// TwinCAT 3 PLC project sACN_PLC
// ProgramVersion: 3.1.4026.18
// libraries:
//   Tc2_Standard, * (Beckhoff Automation GmbH)
//   Tc2_System, * (Beckhoff Automation GmbH)
//   Tc2_TcpIp, * (Beckhoff Automation GmbH)
//   Tc2_Utilities, * (Beckhoff Automation GmbH)
//   Tc3_EventLogger, * (Beckhoff Automation GmbH)
//   Tc3_sACN, * (Beckhoff Automation GmbH)
// project tree:
//   IO/ IO.TcPOU, Term06.TcPOU, Term07.TcPOU
//   / PlcTask.TcTTO
//   POUs/Case_01/ c01_SimpleUsecase.TcPOU
//   POUs/Case_02/ c02_SharingCommunicator.TcPOU
//   POUs/Case_02/SubProgramms/ PRG_SimpleSending.TcPOU, PRG_SimpleReceiving.TcPOU
//   POUs/Case_03/ c03_InteractingWithIO.TcPOU
//   POUs/Case_04/ c4_MultiuniverseSource.TcPOU
//   POUs/Case_05/ c05_CustomFBs.TcPOU
//   POUs/Case_05/SBSPM Extended POUs/ FB_sACN_ReceiverAndMerger_SBSPM.TcPOU, FB_sACN_Source_SBSPM.TcPOU, ST_ReceivedSourceSBSPM.TcDUT
//   POUs/Case_06/ c06_TrackingEvents.TcPOU, FB_sAcnMessagesCatcher.TcPOU
//   POUs/ MAIN.TcPOU
// real-time tasks:
//   TASK PlcTask: cycle T#10ms, priority 20, ADS port 350
// I/O:
//   DEVICE Device 1 (EtherCAT) (disabled), AmsNetId 172.17.152.255.2.1
//     Term 1 (EK1200) [EK1200-5000 EtherCAT Power supply (2A E-Bus)]
//       Term 2 (EK1110) [EK1110 EtherCAT extension]
//     Term 3 (EK1100) [EK1100 EtherCAT Coupler (2A E-Bus)]
//       Term 4 (EL4002) [EL4002 2Ch. Ana. Output 0-10V, 12bit]
//       Term 5 (EL4022) [EL4022 2Ch. Ana. Output 4-20mA, 12bit]
//       Term 6 (EL6851) [EL6851 DMX Master]
//       Term 7 (EL6851-0010) [EL6851-0010 DMX Slave]
//       Term 9 (EL9011) [EL9011 End Terminal]
// variable links:
//   sACN_PLC/sACN_PLC Instance <-> Device 1 (EtherCAT)/Term 3 (EK1100)/Term 6 (EL6851)
//     PlcTask Outputs/Term06.ChannelsLength <-> DMX Control/Channel length
//     PlcTask Outputs/Term06.DmxChannels <-> DMX Channel 1-64/Channel 1
//     PlcTask Outputs/Term06.DmxChannels @bit 72 <-> DMX Channel 1-64/Channel 10
//     PlcTask Outputs/Term06.DmxChannels @bit 80 <-> DMX Channel 1-64/Channel 11
//     PlcTask Outputs/Term06.DmxChannels @bit 88 <-> DMX Channel 1-64/Channel 12
//     PlcTask Outputs/Term06.DmxChannels @bit 96 <-> DMX Channel 1-64/Channel 13
//     PlcTask Outputs/Term06.DmxChannels @bit 104 <-> DMX Channel 1-64/Channel 14
//     PlcTask Outputs/Term06.DmxChannels @bit 112 <-> DMX Channel 1-64/Channel 15
//     PlcTask Outputs/Term06.DmxChannels @bit 120 <-> DMX Channel 1-64/Channel 16
//     PlcTask Outputs/Term06.DmxChannels @bit 8 <-> DMX Channel 1-64/Channel 2
//     PlcTask Outputs/Term06.DmxChannels @bit 16 <-> DMX Channel 1-64/Channel 3
//     PlcTask Outputs/Term06.DmxChannels @bit 24 <-> DMX Channel 1-64/Channel 4
//     PlcTask Outputs/Term06.DmxChannels @bit 32 <-> DMX Channel 1-64/Channel 5
//     PlcTask Outputs/Term06.DmxChannels @bit 40 <-> DMX Channel 1-64/Channel 6
//     PlcTask Outputs/Term06.DmxChannels @bit 48 <-> DMX Channel 1-64/Channel 7
//     PlcTask Outputs/Term06.DmxChannels @bit 56 <-> DMX Channel 1-64/Channel 8
//     PlcTask Outputs/Term06.DmxChannels @bit 64 <-> DMX Channel 1-64/Channel 9
//   sACN_PLC/sACN_PLC Instance <-> Device 1 (EtherCAT)/Term 3 (EK1100)/Term 7 (EL6851-0010)
//     PlcTask Inputs/Term07.DMX_Control_SDX16 <-> DMX Channel 1-64/Channel 1
//     PlcTask Inputs/Term07.DMX_Control_SDX16 @bit 72 <-> DMX Channel 1-64/Channel 10
//     PlcTask Inputs/Term07.DMX_Control_SDX16 @bit 80 <-> DMX Channel 1-64/Channel 11
//     PlcTask Inputs/Term07.DMX_Control_SDX16 @bit 88 <-> DMX Channel 1-64/Channel 12
//     PlcTask Inputs/Term07.DMX_Control_SDX16 @bit 96 <-> DMX Channel 1-64/Channel 13
//     PlcTask Inputs/Term07.DMX_Control_SDX16 @bit 104 <-> DMX Channel 1-64/Channel 14
//     PlcTask Inputs/Term07.DMX_Control_SDX16 @bit 112 <-> DMX Channel 1-64/Channel 15
//     PlcTask Inputs/Term07.DMX_Control_SDX16 @bit 120 <-> DMX Channel 1-64/Channel 16
//     PlcTask Inputs/Term07.DMX_Control_SDX16 @bit 8 <-> DMX Channel 1-64/Channel 2
//     PlcTask Inputs/Term07.DMX_Control_SDX16 @bit 16 <-> DMX Channel 1-64/Channel 3
//     PlcTask Inputs/Term07.DMX_Control_SDX16 @bit 24 <-> DMX Channel 1-64/Channel 4
//     PlcTask Inputs/Term07.DMX_Control_SDX16 @bit 32 <-> DMX Channel 1-64/Channel 5
//     PlcTask Inputs/Term07.DMX_Control_SDX16 @bit 40 <-> DMX Channel 1-64/Channel 6
//     PlcTask Inputs/Term07.DMX_Control_SDX16 @bit 48 <-> DMX Channel 1-64/Channel 7
//     PlcTask Inputs/Term07.DMX_Control_SDX16 @bit 56 <-> DMX Channel 1-64/Channel 8
//     PlcTask Inputs/Term07.DMX_Control_SDX16 @bit 64 <-> DMX Channel 1-64/Channel 9

CONFIGURATION sACN_PLC
    RESOURCE PLC ON TwinCAT3
        TASK PlcTask(INTERVAL := T#10ms, PRIORITY := 20);
        PROGRAM MAIN WITH PlcTask : MAIN;
    END_RESOURCE
END_CONFIGURATION

// ---- POUs/Case_05/SBSPM Extended POUs/ST_ReceivedSourceSBSPM.TcDUT
TYPE ST_ReceivedSourceSBSPM :
STRUCT
	Name 		: STRING(63);
	CID			: Guid;
	Priority	: USINT(0..200);
	IpAddress	: T_IPv4Addr;
	LastFrameNum: USINT;
	SeqErr      : USINT;
	Jumps		: USINT;
	LastPriorities		: ARRAY [1..512] OF USINT;
	LastDMXproperties 	: ARRAY [1..512] OF USINT;
	timeout 	: TON;
END_STRUCT
END_TYPE

// ---- POUs/MAIN.TcPOU
PROGRAM MAIN
VAR
	ChangeValuesTimer : TON;
	i : UINT;
	
	ActiveSample : USINT := 01;
END_VAR

IO();

CASE ActiveSample OF
	01: //<========= CASE 01: Simple Send and Receive sACN Data =========>
		c01_SimpleUsecase();
		
		ChangeValuesTimer(IN:= NOT ChangeValuesTimer.Q, PT:= T#50MS);
		IF ChangeValuesTimer.Q THEN
			FOR i:=1 TO 16 DO
				c01_SimpleUsecase.InDmxData_U111[i] := c01_SimpleUsecase.InDmxData_U111[i] + 1;
				c01_SimpleUsecase.InDmxData_U333[i] := c01_SimpleUsecase.InDmxData_U333[i] - 1;
			END_FOR
		END_IF
	
	02: //<========= CASE 02: Single Communicator, Multiple Subprograms =========>
		c02_SharingCommunicator();
		
	03: //<========= CASE 03: Integration the sACN protocol with hardware DMX terminals =========>
		c03_InteractingWithIO();
		
	04: //<========= CASE 04: Idea for multiuniverse sACN source =========>
		ChangeValuesTimer(IN:= NOT ChangeValuesTimer.Q, PT:= T#50MS);
		
		c4_MultiuniverseSource(	 Enable:= , 
							 SourceName:= 'Sample Multiuniverse Source' ,
									CID:= Tc2_Utilities.STRING_TO_GUID('6f872ff2-8f47-4ea3-a351-549a76e10665')); //Generated by https://www.guidgenerator.com/
									
		IF ChangeValuesTimer.Q THEN
			FOR i:=1 TO 64 DO
				c4_MultiuniverseSource.InDmxData_U111[i] := c4_MultiuniverseSource.InDmxData_U111[i] + 1;
			END_FOR
			FOR i:=1 TO 128 DO
				c4_MultiuniverseSource.InDmxData_U222[i] := c4_MultiuniverseSource.InDmxData_U222[i] - 1;
			END_FOR
			FOR i:=1 TO 256 DO
				c4_MultiuniverseSource.InDmxData_U333[i] := c4_MultiuniverseSource.InDmxData_U333[i] + 1;
			END_FOR
			FOR i:=1 TO 512 DO
				c4_MultiuniverseSource.InDmxData_U444[i] := c4_MultiuniverseSource.InDmxData_U444[i] - 1;
			END_FOR
		END_IF
		
	05: //<========= CASE 05: Castom FB's =========>
		c05_CustomFBs();
END_CASE

//<========= CASE 06: Catching error events =========>
c06_TrackingEvents();

END_PROGRAM

// ---- IO/IO.TcPOU
PROGRAM IO
VAR
END_VAR

Term06();

Term07();

END_PROGRAM

// ---- IO/Term06.TcPOU
//EL6851 Terminal (DMX Master) programm
PROGRAM Term06 
VAR_INPUT
	DmxLightFixture_Left  : ARRAY [1..8] OF USINT;
	DmxLightFixture_Right : ARRAY [1..8] OF USINT;
END_VAR
VAR_OUTPUT
	ChannelsLength	AT %Q*: UINT := 16;
	DmxChannels		AT %Q*: ARRAY [1..16] OF USINT; 
END_VAR

DmxChannels  [1] := DmxLightFixture_Left [1];
DmxChannels  [2] := DmxLightFixture_Left [2];
DmxChannels  [3] := DmxLightFixture_Left [3];
DmxChannels  [4] := DmxLightFixture_Left [4];
                    
DmxChannels  [5] := DmxLightFixture_Left [5];
DmxChannels  [6] := DmxLightFixture_Left [6];
DmxChannels  [7] := DmxLightFixture_Left [7];
DmxChannels  [8] := DmxLightFixture_Left [8];

DmxChannels  [9] := DmxLightFixture_Right [1];
DmxChannels [10] := DmxLightFixture_Right [2];
DmxChannels [11] := DmxLightFixture_Right [3];
DmxChannels [12] := DmxLightFixture_Right [4];
                                                          
DmxChannels [13] := DmxLightFixture_Right [5];
DmxChannels [14] := DmxLightFixture_Right [6];
DmxChannels [15] := DmxLightFixture_Right [7];
DmxChannels [16] := DmxLightFixture_Right [8];

END_PROGRAM

// ---- IO/Term07.TcPOU
//EL6851-0010 Terminal (DMX Slave) programm
PROGRAM Term07
VAR_INPUT
	DMX_Control_SDX16  	AT %I*: ARRAY [1..16] OF USINT;
END_VAR
VAR_OUTPUT
	DmxArrayTo_sAcn_U111 : ARRAY [1..16] OF USINT;
END_VAR

DmxArrayTo_sAcn_U111[01] := DMX_Control_SDX16[01];
DmxArrayTo_sAcn_U111[02] := DMX_Control_SDX16[02];
DmxArrayTo_sAcn_U111[03] := DMX_Control_SDX16[03];
DmxArrayTo_sAcn_U111[04] := DMX_Control_SDX16[04];
DmxArrayTo_sAcn_U111[05] := DMX_Control_SDX16[05];
DmxArrayTo_sAcn_U111[06] := DMX_Control_SDX16[06];
DmxArrayTo_sAcn_U111[07] := DMX_Control_SDX16[07];
DmxArrayTo_sAcn_U111[08] := DMX_Control_SDX16[08];

DmxArrayTo_sAcn_U111[09] := DMX_Control_SDX16[09];
DmxArrayTo_sAcn_U111[10] := DMX_Control_SDX16[10];
DmxArrayTo_sAcn_U111[11] := DMX_Control_SDX16[11];
DmxArrayTo_sAcn_U111[12] := DMX_Control_SDX16[12];
DmxArrayTo_sAcn_U111[13] := DMX_Control_SDX16[13];
DmxArrayTo_sAcn_U111[14] := DMX_Control_SDX16[14];
DmxArrayTo_sAcn_U111[15] := DMX_Control_SDX16[15];
DmxArrayTo_sAcn_U111[16] := DMX_Control_SDX16[16];

END_PROGRAM

// ---- POUs/Case_01/c01_SimpleUsecase.TcPOU
PROGRAM c01_SimpleUsecase
VAR_INPUT
	Enable : BOOL; //Boolean input to enable the receivers
	InDmxData_U111 : ARRAY [1..16] OF USINT; //Arrays containing the DMX data to be sent to universe 111
	InDmxData_U333 : ARRAY [1..16] OF USINT; //Arrays containing the DMX data to be sent to universe 333
END_VAR
VAR_OUTPUT
	isInited 		: BOOL; //Indicates if the initialization is complete.
	OutDmxData_U222 : ARRAY [1..16] OF USINT; //Array to store the DMX data for universes 222
	OutDmxData_U444 : ARRAY [1..16] OF USINT; //Array to store the DMX data for universes 444
END_VAR
VAR
	sACN_Com : FB_sACN_UDP_Communicator;
	
	sACN_Sender_U111: FB_sACN_Source;
	sACN_Sender_U333: FB_sACN_SourceExtDmx;
	
	sACN_Receiver_U222:	FB_sACN_Receiver;
	sACN_Receiver_U444:	FB_sACN_ReceiverAndMerger;

	LastReceivedPacketNum : UINT;
	i : UINT;
END_VAR

sACN_Com(NetworkAdapterNum:= E_NetworkAdapters.SLOT_N02, //<- Change NIC here if it is necessary
			 ReconnectTime:= T#5M, 
			 BindedToNetworkAdapter=> , 
			 BindedAdapterInfo=> );

// Direct Assignment Approach: Assign DMX channel values directly without binding.
sACN_Sender_U111(
	sAcnCommunicator:= sACN_Com,
	Enable:= Enable,
	SourceName:= 'BeckhoffPLC sACN Source 111',
	CID:= Tc2_Utilities.STRING_TO_GUID('3566cea5-b4a4-48fc-aa02-cd84a65f0a88'), //Generated by https://www.guidgenerator.com/
	sAcnUniverse:= 111,
	PacketPriority:= 90,
	SendingPeriod:= T#40MS,
	DmxChannels:= ,
	SentPackets=> );
	
FOR i:=1 TO 16 DO
	sACN_Sender_U111.DmxChannels[i] := InDmxData_U111[i];
END_FOR

//Packet Extraction Approach: Extract DMX data upon receiving a new packet.
sACN_Receiver_U222(
	sAcnCommunicator:= sACN_Com, 
	Enable			:= Enable,
	sAcnUniverse	:= 222);

IF sACN_Receiver_U222.ReceiveCounter <> LastReceivedPacketNum THEN // A new sACN packet has been received.
	LastReceivedPacketNum := sACN_Receiver_U222.ReceiveCounter;
	
	// Check if the received packet is a data packet.
	IF  sACN_Receiver_U222.ReceivedPacket.AsDataPacket.FL02_VectorFraming = Tc3_sACN.sACN_Params.VECTOR_E131_DATA_PACKET THEN
		// Extract and store DMX data from the received packet.
		FOR i:=1 TO 16 DO
			OutDmxData_U222[i] := sACN_Receiver_U222.ReceivedPacket.AsDataPacket.DL07_PropertyValues[i+1];
		END_FOR
	END_IF
END_IF

// Direct Binding Approach: Bind the external DMX data array for universe 444 to allow direct manipulation of the received values.
IF NOT isInited THEN
	// Bind the external DMX data array for universe 444 to allow direct manipulation of the received values.
	sACN_Sender_U333.BindExternalDmxArray(InDmxData_U333);
	sACN_Receiver_U444.BindExternalDmxArray(OutDmxData_U444);
	isInited := TRUE;
END_IF	 

sACN_Sender_U333(
	sAcnCommunicator:= sACN_Com, 
	Enable:= Enable, 
	SourceName:= 'BeckhoffPLC sACN Source 333', 
	CID:= Tc2_Utilities.STRING_TO_GUID('767c315b-0c1d-4851-b956-6a6cce014b93'), //Generated by https://www.guidgenerator.com/
	sAcnUniverse:= 333, 
	PacketPriority:= 95, 
	SendingPeriod:= T#50MS, 
	SentPackets=> );

sACN_Receiver_U444(
	sAcnCommunicator:= sACN_Com, 
	Enable			:= Enable, 
	sAcnUniverse	:= 444, 
	MergeRule		:= E_DmxMergeRules.HVP);

END_PROGRAM

// ---- POUs/Case_02/c02_SharingCommunicator.TcPOU
PROGRAM c02_SharingCommunicator
VAR
	sACN_Com : FB_sACN_UDP_Communicator;
	
	ChangeValuesTimer : TON;
	i : UINT;
END_VAR

sACN_Com(NetworkAdapterNum:= E_NetworkAdapters.SLOT_N02, //<- Change if it is necessary
			 ReconnectTime:= T#5M, 
			 BindedToNetworkAdapter=> , 
			 BindedAdapterInfo=> );
			 
PRG_SimpleReceiving(
	sACN_ExternalCommunicator:= sACN_Com, 
	Enable:= , 
	isInited=> , 
	OutDmxData_U222=> , 
	OutDmxData_U444=> );
	
FOR i:=1 TO 16 DO
	PRG_SimpleSending.InDmxData_U111[i] := PRG_SimpleSending.InDmxData_U111[i] + 1;
	PRG_SimpleSending.InDmxData_U333[i] := PRG_SimpleSending.InDmxData_U333[i] - 1;
END_FOR

PRG_SimpleSending(
	Enable:= , 
	sACN_ExternalCommunicator:= sACN_Com, 
	InDmxData_U111:= , 
	InDmxData_U333:= , 
	isInited=> );

END_PROGRAM

// ---- POUs/Case_02/SubProgramms/PRG_SimpleReceiving.TcPOU
PROGRAM PRG_SimpleReceiving
VAR_INPUT
	sACN_ExternalCommunicator : Tc3_sACN.I_sAcnCommunicator;
	Enable : BOOL; //Boolean input to enable the receivers
END_VAR
VAR_OUTPUT
	isInited 		: BOOL; //Indicates if the initialization is complete.
	OutDmxData_U222 : ARRAY [1..16] OF USINT; //Array to store the DMX data for universes 222
	OutDmxData_U444 : ARRAY [1..16] OF USINT; //Array to store the DMX data for universes 444
END_VAR
VAR
	sACN_Receiver_U222:	Tc3_sACN.FB_sACN_Receiver;
	sACN_Receiver_U444:	Tc3_sACN.FB_sACN_ReceiverAndMerger;
	
	LastReceivedPacketNum : UINT;
	i : UINT;
END_VAR

IF sACN_ExternalCommunicator <> 0 THEN
//Packet Extraction Approach: Extract DMX data upon receiving a new packet.
	sACN_Receiver_U222(
		sAcnCommunicator:= sACN_ExternalCommunicator, 
		Enable			:= Enable,
		sAcnUniverse	:= 222);
	
	IF sACN_Receiver_U222.ReceiveCounter <> LastReceivedPacketNum THEN // A new sACN packet has been received.
		LastReceivedPacketNum := sACN_Receiver_U222.ReceiveCounter;
		
		// Check if the received packet is a data packet.
		IF  sACN_Receiver_U222.ReceivedPacket.AsDataPacket.FL02_VectorFraming = Tc3_sACN.sACN_Params.VECTOR_E131_DATA_PACKET THEN
			// Extract and store DMX data from the received packet.
			FOR i:=1 TO 16 DO
				OutDmxData_U222[i] := sACN_Receiver_U222.ReceivedPacket.AsDataPacket.DL07_PropertyValues[i+1];
			END_FOR
		END_IF
	END_IF
	
// Direct Binding Approach: Bind the external DMX data array for universe 444 to allow direct manipulation of the received values.
	IF NOT isInited THEN
		// Bind the external DMX data array for universe 444 to allow direct manipulation of the received values.
		sACN_Receiver_U444.BindExternalDmxArray(OutDmxData_U444);
		isInited := TRUE;
	END_IF	 
	
	sACN_Receiver_U444(
		sAcnCommunicator:= sACN_ExternalCommunicator, 
		Enable			:= Enable, 
		sAcnUniverse	:= 444, 
		MergeRule		:= E_DmxMergeRules.HVP);
END_IF

END_PROGRAM

// ---- POUs/Case_02/SubProgramms/PRG_SimpleSending.TcPOU
PROGRAM PRG_SimpleSending
VAR_INPUT
	Enable 			: BOOL; //Boolean input to enable the receivers
	sACN_ExternalCommunicator : Tc3_sACN.I_sAcnCommunicator;
	InDmxData_U111 : ARRAY [1..16] OF USINT; //Arrays containing the DMX data to be sent to universe 111
	InDmxData_U333 : ARRAY [1..16] OF USINT; //Arrays containing the DMX data to be sent to universe 333
END_VAR
VAR_OUTPUT
	isInited : BOOL; //Indicates if the initialization is complete.
END_VAR
VAR
	sACN_Sender_U111: FB_sACN_Source;
	sACN_Sender_U333: FB_sACN_SourceExtDmx;

	i : UINT;
END_VAR

// Direct Assignment Approach: Assign DMX channel values directly without binding.
sACN_Sender_U111(
	sAcnCommunicator:= sACN_ExternalCommunicator, 
	Enable:= Enable, 
	SourceName:= 'BeckhoffPLC sACN Source 111', 
	CID:= Tc2_Utilities.STRING_TO_GUID('3566cea5-b4a4-48fc-aa02-cd84a65f0a88'),  //Generated by https://www.guidgenerator.com/
	sAcnUniverse:= 111, 
	PacketPriority:= 90, 
	SendingPeriod:= T#40MS, 
	DmxChannels:= , 
	SentPackets=> );
	
FOR i:=1 TO 16 DO
	sACN_Sender_U111.DmxChannels[i] := InDmxData_U111[i];
END_FOR

// Binding Approach: Bind external DMX data array for automatic handling.
IF NOT isInited THEN
	sACN_Sender_U333.BindExternalDmxArray(InDmxData_U333);
	isInited := TRUE;
END_IF
	
sACN_Sender_U333(
	sAcnCommunicator:= sACN_ExternalCommunicator, 
	Enable:= Enable, 
	SourceName:= 'BeckhoffPLC sACN Source 333', 
	CID:= Tc2_Utilities.STRING_TO_GUID('767c315b-0c1d-4851-b956-6a6cce014b93'), //Generated by https://www.guidgenerator.com/
	sAcnUniverse:= 333, 
	PacketPriority:= 95, 
	SendingPeriod:= T#50MS, 
	SentPackets=> );

END_PROGRAM

// ---- POUs/Case_03/c03_InteractingWithIO.TcPOU
PROGRAM c03_InteractingWithIO
VAR_INPUT
	Enable 			: BOOL;
END_VAR
VAR_OUTPUT
	isInited : BOOL;
END_VAR
VAR
	sACN_Com : FB_sACN_UDP_Communicator;
		
	sACN_Sender_U111: FB_sACN_SourceExtDmx;
	
	sACN_Receiver_U222:	FB_sACN_Receiver;
	sACN_Receiver_U444:	FB_sACN_ReceiverAndMerger;
	
	LastReceivedPacketNum : UINT;
	i : UINT;
END_VAR

IF NOT isInited THEN
	sACN_Sender_U111.BindExternalDmxArray(Term07.DmxArrayTo_sAcn_U111);
	//sACN_Receiver_U444.BindExternalDmxArray(Term06.DmxLightFixture_Left);
	isInited := TRUE;
END_IF

CallAllFbs(); //with graphical representation of Fbs
	 
IF sACN_Receiver_U222.ReceiveCounter <> LastReceivedPacketNum THEN//New sACN Packet has been received
	LastReceivedPacketNum := sACN_Receiver_U222.ReceiveCounter;
	//Demonstration of how to extract and utilize DMX data from received packets.
	//You alwayes have a direct access to a recieved packete. sACN_Receiver_U444.ReceiveCounter varible can show you if you got the new one.
	IF  sACN_Receiver_U222.ReceivedPacket.AsDataPacket.FL02_VectorFraming = Tc3_sACN.sACN_Params.VECTOR_E131_DATA_PACKET THEN //Received sACN Packet is Data Packet
		FOR i:=1 TO 8 DO
			Term06.DmxLightFixture_Left[i] := sACN_Receiver_U222.ReceivedPacket.AsDataPacket.DL07_PropertyValues[i+1];
			Term06.DmxLightFixture_Right[i]:= sACN_Receiver_U222.ReceivedPacket.AsDataPacket.DL07_PropertyValues[8 + i+1];
		END_FOR
	END_IF
END_IF

ACTION CallAllFbs:
sACN_Com(NetworkAdapterNum := E_NetworkAdapters.SLOT_N01, ReconnectTime := T#5M); // FB_sACN_UDP_Communicator
sACN_Sender_U111(
    sAcnCommunicator := sACN_Com,
    Enable := Enable,
    SourceName := 'sACN Source U111 ShowCase03',
    CID := Tc2_Utilities.STRING_TO_GUID('a3871605-ff16-48b4-b569-d1b9cc2e14dc'),
    sAcnUniverse := 111,
    PacketPriority := 100,
    SendingPeriod := T#100ms); // Tc3_sACN.FB_sACN_SourceExtDmx
sACN_Receiver_U222(sAcnCommunicator := sACN_Com, Enable := Enable, sAcnUniverse := 222); // FB_sACN_Receiver
sACN_Receiver_U444(
    sAcnCommunicator := sACN_Com,
    Enable := Enable,
    sAcnUniverse := 444,
    MergeRule := E_DmxMergeRules.LVP); // Tc3_sACN.FB_sACN_ReceiverAndMerger
END_ACTION

END_PROGRAM

// ---- POUs/Case_04/c4_MultiuniverseSource.TcPOU
PROGRAM c4_MultiuniverseSource
VAR_INPUT
	Enable : BOOL;
	SourceName: STRING(63);
	CID: GUID; 
	
	InDmxData_U111 : ARRAY [1..64] OF USINT; //Arrays containing the DMX data to be sent to universe 111
	InDmxData_U222 : ARRAY [1..128] OF USINT; //Arrays containing the DMX data to be sent to universe 333
	InDmxData_U333 : ARRAY [1..256] OF USINT; //Arrays containing the DMX data to be sent to universe 111
	InDmxData_U444 : ARRAY [1..512] OF USINT; //Arrays containing the DMX data to be sent to universe 333
END_VAR
VAR_OUTPUT
	isInited : BOOL;
END_VAR
VAR
	sACN_Com : FB_sACN_UDP_Communicator;
	
	sACN_Sender_U111: FB_sACN_Source;
	sACN_Sender_U222: FB_sACN_SourceExtDmx;
	sACN_Sender_U333: FB_sACN_Source;
	sACN_Sender_U444: FB_sACN_SourceExtDmx;
	
	i : UINT;
END_VAR

IF NOT isInited THEN
	// Bind the external DMX data array for universe 444 to allow direct manipulation of the received values.
	sACN_Sender_U222.BindExternalDmxArray(InDmxData_U222);
	sACN_Sender_U444.BindExternalDmxArray(InDmxData_U444);
	isInited := TRUE;
END_IF

sACN_Com(NetworkAdapterNum:= E_NetworkAdapters.SLOT_N02, //<- Change if it is necessary
			 ReconnectTime:= T#5M, 
			 BindedToNetworkAdapter=> , 
			 BindedAdapterInfo=> );	

sACN_Sender_U111(
	sAcnCommunicator:= sACN_Com, 
	Enable:= Enable, 
	SourceName:= SourceName, 
	CID:= CID, 
	sAcnUniverse:= 111, 
	PacketPriority:= , 
	SendingPeriod:= , 
	DmxChannels:= , 
	SentPackets=> );

FOR i:=1 TO 64 DO
	sACN_Sender_U111.DmxChannels[i] := InDmxData_U111[i];
END_FOR
	
sACN_Sender_U222(
	sAcnCommunicator:= sACN_Com, 
	Enable:= Enable, 
	SourceName:= SourceName, 
	CID:= CID, 
	sAcnUniverse:= 222, 
	PacketPriority:= , 
	SendingPeriod:= , 
	SentPackets=> );
	
sACN_Sender_U333(
	sAcnCommunicator:= sACN_Com, 
	Enable:= Enable, 
	SourceName:= SourceName, 
	CID:= CID, 
	sAcnUniverse:= 333, 
	PacketPriority:= , 
	SendingPeriod:= , 
	DmxChannels:= , 
	SentPackets=> );
	
FOR i:=1 TO 256 DO
	sACN_Sender_U333.DmxChannels[i] := InDmxData_U333[i];
END_FOR
	
sACN_Sender_U444(
	sAcnCommunicator:= sACN_Com, 
	Enable:= Enable, 
	SourceName:= SourceName, 
	CID:= CID, 
	sAcnUniverse:= 444, 
	PacketPriority:= , 
	SendingPeriod:= , 
	SentPackets=> );

END_PROGRAM

// ---- POUs/Case_05/c05_CustomFBs.TcPOU
PROGRAM c05_CustomFBs
VAR_INPUT
	Enable 			: BOOL;
END_VAR
VAR_OUTPUT
	isInited : BOOL;
END_VAR
VAR
	sACN_Com : FB_sACN_UDP_Communicator; //Transit variable representing the UDP communicator for sACN.

	sACN_Sender_U111: FB_sACN_Source_SBSPM;//Custom Functionality FB
	
	sACN_Receiver_U555:	FB_sACN_ReceiverAndMerger_SBSPM;
	
	LastReceivedPacketNum : UINT;
	i : UINT;
END_VAR

sACN_Com(NetworkAdapterNum:= E_NetworkAdapters.SLOT_N02, //<- Change if it is necessary
			 ReconnectTime:= T#5M, 
			 BindedToNetworkAdapter=> , 
			 BindedAdapterInfo=> );
			 
IF NOT isInited THEN
	isInited := TRUE;
	
	sACN_Receiver_U555.BindExternalDmxArray(Term06.DmxLightFixture_Left);
END_IF

sACN_Sender_U111(
	sAcnCommunicator:= sACN_Com, 
	Enable:= Enable, 
	SourceName:= 'BeckhoffPLC ControlPanel U111', 
	CID:= Tc2_Utilities.STRING_TO_GUID('3566cea5-b4a4-48fc-aa02-cd84a65f0a88'),  //Generated by https://www.guidgenerator.com/
	sAcnUniverse:= 111, 
	PacketPriority:= 100, 
	SendingPeriod:= T#100MS, 
	SentPackets=> );

sACN_Receiver_U555(
	sAcnCommunicator:= sACN_Com, 
	Enable:= Enable,
	sAcnUniverse:= 555,
	MergeRule:= );

END_PROGRAM

// ---- POUs/Case_05/SBSPM Extended POUs/FB_sACN_Source_SBSPM.TcPOU
//Slot-By-Slot Priority Mode
//A variation of this uses DMX512-A START Code DDh (see [DMX] and http://tsp.esta.org/tsp/working_groups/CP/DMXAlternateCodes.php) 
//to indicate slot-by-slot priority before merging the highest priority data for each slot on an HTP basis.
FUNCTION_BLOCK FB_sACN_Source_SBSPM EXTENDS FB_sACN_Source
VAR_INPUT
	DmxPrioriries : ARRAY [1..512] OF USINT;
END_VAR

SUPER^();

METHOD WriteDataPacket : BOOL
VAR_IN_OUT
	packet	: Tc3_sACN.U_sACN_Packet;
END_VAR
VAR_STAT
	wtPriorPacket : BOOL;// is current packet a packet with priorities&
	i : DINT;
END_VAR
SUPER^.WriteDataPacket(packet:=packet);

IF wtPriorPacket THEN
	packet.AsDataPacket.DL07_PropertyValues[1] := 16#DD;
	FOR i := 1 TO 512 DO
		packet.AsDataPacket.DL07_PropertyValues[i+1] := DmxPrioriries[i];
	END_FOR
END_IF

wtPriorPacket := NOT wtPriorPacket;
END_METHOD

END_FUNCTION_BLOCK

// ---- POUs/Case_05/SBSPM Extended POUs/FB_sACN_ReceiverAndMerger_SBSPM.TcPOU
{attribute 'hide_all_locals'}
FUNCTION_BLOCK FB_sACN_ReceiverAndMerger_SBSPM EXTENDS FB_sACN_Receiver
VAR_INPUT
	MergeRule		: E_DmxMergeRules := E_DmxMergeRules.LVP;//Rule for merging DMX values from multiple sources. Default is set to LVP (Latest Value Priority).
END_VAR
VAR_OUTPUT
	ActiveSources 	: ARRAY [1..sACN_Params.MAX_RECEIVED_SOURCES] OF ST_ReceivedSourceSBSPM;//Array holding information about active sources currently being received.
END_VAR
VAR

END_VAR

SUPER^();

CheckExeededActiveSources();

//Iterates through active sources and checks for timeouts. 
//If a timeout occurs, it logs the event and removes the source from the list.
METHOD PROTECTED CheckExeededActiveSources : BOOL
VAR
	i : UINT;
END_VAR
FOR i:=1 TO sACN_Params.MAX_RECEIVED_SOURCES DO
	IF ActiveSources[i].Name <> '' THEN
		ActiveSources[i].timeout(IN := TRUE, PT := sACN_Params.SACN_RECEIVER_TIMEOUT);
		IF ActiveSources[i].timeout.Q THEN
			_logger.Log_sACN_Receiver_DeleteSource(sAcnUniverse, ActiveSources[i].Name, ActiveSources[i].timeout.PT);		
			ForgetSource(i);
		END_IF
	END_IF
END_FOR
END_METHOD

//Removes a source from the active sources list by shifting the remaining sources up in the array. 
//If all sources are gone, it calls OnAllActiveSourcesAreGone
METHOD PROTECTED ForgetSource : BOOL
VAR_INPUT
	SourceNum: UINT; //
END_VAR
VAR
	i : UINT;
	emptySource : ST_ReceivedSourceSBSPM;
END_VAR
IF SourceNum > 0 AND SourceNum <= sACN_Params.MAX_RECEIVED_SOURCES THEN
	FOR i:=SourceNum TO sACN_Params.MAX_RECEIVED_SOURCES DO
		IF i <> sACN_Params.MAX_RECEIVED_SOURCES THEN
			ActiveSources[i] := ActiveSources[i+1];
		ELSE
			ActiveSources[i] := emptySource;
		END_IF
	END_FOR
END_IF

FOR i:=1 TO sACN_Params.MAX_RECEIVED_SOURCES DO
	IF ActiveSources[i].Name <> '' THEN
		RETURN;
	END_IF
END_FOR

OnAllActiveSourcesAreGone();
END_METHOD

//Checks if a source is known and updates its priority and sequence number, logging any sequence errors
METHOD PROTECTED GetReceivedSourceNumber : UINT
VAR_IN_OUT
	Source: ST_ReceivedSourceSBSPM;
END_VAR
VAR
	i : UINT;
END_VAR
FOR i:=1 TO sACN_Params.MAX_RECEIVED_SOURCES DO
	IF Tc3_Module.GuidsEqual(ADR(ActiveSources[i].CID), ADR(Source.CID)) THEN
		ActiveSources[i].Priority := Source.Priority;
		
		IF (Source.LastFrameNum - ActiveSources[i].LastFrameNum) > 1 AND_THEN
		  (Source.LastFrameNum <> 1 AND ActiveSources[i].LastFrameNum <> 255) THEN
			ActiveSources[i].SeqErr := ActiveSources[i].SeqErr + 1;
			ActiveSources[i].Jumps := Source.LastFrameNum - ActiveSources[i].LastFrameNum;
		END_IF
		
		ActiveSources[i].LastFrameNum := Source.LastFrameNum;
		
		ActiveSources[i].timeout(IN := FALSE);
		
		GetReceivedSourceNumber := i;
		RETURN;
	END_IF
END_FOR
END_METHOD

METHOD PROTECTED MergeToExternalDmxArray : BOOL
VAR_INPUT
END_VAR
VAR_STAT
	i, j 			: DINT;
	temp_val: USINT;
	temp_num :DINT ;
END_VAR
IF _extNum > 0 AND _extNum <= 512 THEN
	FOR i:= 1 TO _extNum DO
		temp_val := 0;
		temp_num := 1;
		FOR j:=1 TO sACN_Params.MAX_RECEIVED_SOURCES DO
			IF ActiveSources[j].LastPriorities[i] > temp_val THEN
				temp_val := ActiveSources[j].LastPriorities[i];
				temp_num := j;
			END_IF
		_externalDmxArray[i]^ := ActiveSources[temp_num].LastDMXproperties[i];
		END_FOR
	END_FOR
END_IF
END_METHOD

//Clears the received packet and resets the external DMX array when no active sources are left.
METHOD PROTECTED OnAllActiveSourcesAreGone : BOOL
VAR
	i : DINT;
	emptyDataPacket : ST_SACN_DataPacket;
END_VAR
ReceivedPacket.AsDataPacket := emptyDataPacket;

IF _extNum > 0 AND _extNum <= 512 THEN
	FOR i:= 1 TO _extNum DO
		_externalDmxArray[i]^:= 0;
	END_FOR
END_IF
END_METHOD

METHOD OnSAcnDataPacketReceived : BOOL
VAR_IN_OUT
	Packet 			: ST_SACN_DataPacket;
END_VAR
VAR_INPUT
	sRemoteHost : T_IPv4Addr ;
END_VAR
VAR
	i, j 			: DINT;
	SenderNum		: DINT;
	temp_val: USINT;
	temp_num :DINT ;
	gotSamePriority : USINT;
	currentSource	: ST_ReceivedSourceSBSPM;
END_VAR
SUPER^.OnSAcnDataPacketReceived(Packet, sRemoteHost);

currentSource.Name 			:= Packet.FL03_SourceName.AsString;
currentSource.Priority  	:= Packet.FL04_Priority;
currentSource.CID 			:= Packet.RL06_CID;
currentSource.IpAddress 	:= sRemoteHost;
currentSource.LastFrameNum 	:= Packet.FL06_SequenceNumber;

SenderNum := GetReceivedSourceNumber(currentSource);

IF SenderNum = 0 THEN //if known update data inside method _isReceivedSourceKnown
	SenderNum := SaveSource(currentSource);	
END_IF

IF Packet.DL07_PropertyValues[1] = 16#00 THEN
	FOR i := 1 TO 512 DO//Update DMX Array in ActiveSource
		ActiveSources[SenderNum].LastDMXproperties[i] := Packet.DL07_PropertyValues[i+1];
	END_FOR
ELSIF Packet.DL07_PropertyValues[1] = 16#DD THEN
	FOR i := 1 TO 512 DO//Update Priority Array in ActiveSource
		ActiveSources[SenderNum].LastPriorities[i] := Packet.DL07_PropertyValues[i+1];
	END_FOR
END_IF

MergeToExternalDmxArray();
END_METHOD

//Saves a new source to the list of active sources if there is an empty slot available. Logs the event upon saving
//Returns the number of stored element in ActiveSources array.
METHOD PRIVATE SaveSource : UINT
VAR_IN_OUT
	Source: ST_ReceivedSourceSBSPM;
END_VAR
VAR
	i : UINT;
END_VAR
FOR i:=1 TO sACN_Params.MAX_RECEIVED_SOURCES DO
	IF ActiveSources[i].Name = '' THEN
		_logger.Log_sACN_Receiver_SaveSource(sAcnUniverse, Source.Name);

		ActiveSources[i] := Source;
		SaveSource := i;
		RETURN;
	END_IF
END_FOR
END_METHOD

END_FUNCTION_BLOCK

// ---- POUs/Case_06/c06_TrackingEvents.TcPOU
PROGRAM c06_TrackingEvents
VAR
	sAcnLibEventsHandler  : FB_sAcnMessagesCatcher;// Extended instance of the event catcher. 
	// Monitors sACN receiver events and counts Enabled/Disabled transitions for the configured universe
END_VAR

// In the example, the application monitors the OnSACN_Receiver_Disabled and OnSACN_Receiver_Enabled events. 
// FB_sAcnMessagesCatcher override the methods provided by FB_sAcnLibEventsCatcher and implement the actions your application should take. 
// The base class defines these methods and wires the events for you.
// your overrides add the custom behavior while the catcher handles the rest.

sAcnLibEventsHandler(sAcnReceiverUniverse		:= 222, 
					RecieverEnabledEventsCount	=> , 
					RecieverDisabledEventsCount	=> );

END_PROGRAM

// ---- POUs/Case_06/FB_sAcnMessagesCatcher.TcPOU
//When you need to react to events in code, you can catch them directly in your application 
//by inheriting from FB_sAcnLibEventsCatcher. This base component already implements the event 
//subscription and dispatch logic, so the approach is context‑independent and requires no additional configuration.
FUNCTION_BLOCK FB_sAcnMessagesCatcher EXTENDS FB_sAcnLibEventsCatcher
VAR_INPUT
	sAcnReceiverUniverse 		: UINT;// Target sACN universe number to monitor. Events are filtered for this universe
END_VAR
VAR_OUTPUT
	RecieverEnabledEventsCount 	: UINT;// Count of OnSACN_Receiver_Enabled events observed for the selected universe
	RecieverDisabledEventsCount : UINT;// Count of OnSACN_Receiver_Disabled events observed for the selected universe
END_VAR
VAR
END_VAR

// Call the parent implementation to keep default logging/event binding from FB_sAcnLibEventsCatcher
SUPER^();SUPER^();

//JSON ATTRIBUTE : {sAcnUniverse : [UINT]}
METHOD OnSACN_Receiver_Disabled : BOOL
VAR_INPUT
    fbEvent : REFERENCE TO FB_TcEvent;
END_VAR
VAR
	sAcnUniverse : UINT;
END_VAR
// Each event handler method can include attributes that carry extra information about the event.
// The available attributes are documented in the method’s comment header as a JSON descriptor 
// (for example, //JSON ATTRIBUTE : {sAcnUniverse : [UINT]}). To read these values at runtime, 
// use ParseJsonAttributeFromEvent, which extracts an attribute by name from the FB_TcEvent into your variable. 
// The example shown retrieves the sAcnUniverse attribute and then uses it to filter and count the relevant events.

THIS^.ParseJsonAttributeFromEvent(fbEvent, 'sAcnUniverse', sAcnUniverse);

IF sAcnUniverse = sAcnReceiverUniverse THEN
	RecieverDisabledEventsCount := RecieverDisabledEventsCount + 1;
END_IF
END_METHOD

//JSON ATTRIBUTE : {sAcnUniverse : [UINT]}
METHOD OnSACN_Receiver_Enabled : BOOL
VAR_INPUT
    fbEvent : REFERENCE TO FB_TcEvent;
END_VAR
VAR
	sAcnUniverse : UINT;
END_VAR
// Each event handler method can include attributes that carry extra information about the event.
// The available attributes are documented in the method’s comment header as a JSON descriptor 
// (for example, //JSON ATTRIBUTE : {sAcnUniverse : [UINT]}). To read these values at runtime, 
// use ParseJsonAttributeFromEvent, which extracts an attribute by name from the FB_TcEvent into your variable. 
// The example shown retrieves the sAcnUniverse attribute and then uses it to filter and count the relevant events.

THIS^.ParseJsonAttributeFromEvent(fbEvent, 'sAcnUniverse', sAcnUniverse);

IF sAcnUniverse = sAcnReceiverUniverse THEN
	RecieverEnabledEventsCount := RecieverEnabledEventsCount + 1;
END_IF
END_METHOD

END_FUNCTION_BLOCK
